# B&R Automation Studio project template1
Automation Studio 4.5.2.102

## Configuration Config1

### IoMap.iom - 4PP065_0571_P74/IoMap.iom
```iecst
VAR_CONFIG
	Cyclic#1.gAxis01_DrvIf.iLifeCnt AT %IB."8I64xxxxxxx.00x-1".SDC_LifeCnt;
	Cyclic#1.gAxis01_DrvIf.iDrvOK AT %IX."8I64xxxxxxx.00x-1".ETAD_Input_Bool_02;
	Cyclic#1.gAxis01_DrvIf.oSetTime AT %QW."8I64xxxxxxx.00x-1".SDC_SetTime;
	Cyclic#1.::speed AT %QW."8I64xxxxxxx.00x-1".LFRD_Output;
	Cyclic#1.gAxis01_DiDoIf.iLifeCntDriveReady AT %IB."8I64xxxxxxx.00x-1".SDC_LifeCnt;
	Cyclic#1.gAxis01_DiDoIf.iLifeCntDriveEnable AT %IB."8I64xxxxxxx.00x-1".SDC_LifeCnt;
	Cyclic#1.gAxis01_DiDoIf.oDriveEnable AT %QX."8I64xxxxxxx.00x-1".CMDD_Output_Bool_00;
	Cyclic#1.gAxis01_ModuleOk AT %QX."8I64xxxxxxx.00x-1".CMDD_Output_Bool_01;
	Cyclic#1.gAxis01_ModuleOk AT %QX."8I64xxxxxxx.00x-1".CMDD_Output_Bool_02;
	Cyclic#1.gAxis01_ModuleOk AT %IX."8I64xxxxxxx.00x-1".ModuleOk;
	Cyclic#1.gAxis01_DiDoIf.oDriveEnable AT %QX."8I64xxxxxxx.00x-1".CMDD_Output_Bool_03;
	Cyclic#1.gAxis01_DiDoIf.iDriveReady AT %IX."8I64xxxxxxx.00x-1".ETAD_Input_Bool_02;
	::EVIRD.STATE AT %IW."8I64xxxxxxx.00x-1".ETAD_Input;
	::EVIRD.CMD AT %QW."8I64xxxxxxx.00x-1".CMDD_Output;
	::led1 AT %QX."X20DO9322".DigitalOutput02;
	::led2 AT %QX."X20DO9322".DigitalOutput03;
	::led3 AT %QX."X20DO9322".DigitalOutput04;
	::led4 AT %QX."X20DO9322".DigitalOutput05;
	::real_speed AT %IW."8I64xxxxxxx.00x-1".RFRD_Input;
END_VAR
```

## Logical view

### Global.var
```iecst
VAR
	gAxis01 : ACP10AXIS_typ;
	gAxis01_HW : SdcHwCfg_typ := (0);
	gAxis01_DrvIf : SdcDrvIf16_typ := (0);
	gAxis01_DiDoIf : SdcDiDoIf_typ := (0);
	gAxis01_ModuleOk : BOOL := 0;
	speed : INT := 500;
	EVIRD : DRIVE;
	start : INT := 0;
	Button_1 : BOOL;
	led : ARRAY[0..3] OF BOOL;
	led4 : BOOL;
	led3 : BOOL;
	led2 : BOOL;
	led1 : BOOL;
	Button_3 : BOOL;
	Button_2 : BOOL;
	Button_4 : BOOL;
	real_speed : {REDUND_UNREPLICABLE} INT;
END_VAR
```

- Visualisation Logical/gAxis01obj/Visu (not shown)

### Library Logical/Libraries/Library

#### Library.fun
```iecst
{REDUND_ERROR} FUNCTION_BLOCK DRIVE (*TODO: Add your comment here*) (*$GROUP=User,$CAT=User,$GROUPICON=User.png,$CATICON=User.png*)
	VAR_INPUT
		ENABLED : BOOL;
		STATE : UINT;
	END_VAR
	VAR_OUTPUT
		CMD : UINT;
	END_VAR
END_FUNCTION_BLOCK
```

#### DRIVE.c
```c
#include <bur/plctypes.h>
#ifdef __cplusplus
	extern "C"
	{
#endif
	#include "Library.h"
#ifdef __cplusplus
	};
#endif
/* TODO: Add your comment here */
void DRIVE(struct DRIVE* inst)
{
	UINT mask= inst->STATE & 0x6f;
	if(!inst->ENABLED)
	{
		inst->CMD =CMD_SHUTDOWN;
	}
	else
	{
		switch(mask)
		{
			case STATE_DISABLED:
				inst->CMD=CMD_SHUTDOWN;
				break;
			case STATE_READY:
				inst->CMD=CMD_ENABLED;
				break;
			case STATE_SWITCHED_ON:
				inst->CMD=CMD_SWITCHED_ON;
				break;
		}
	}
}
```

### Program Logical/Program

#### Main.c
```c
#include <bur/plctypes.h>

#ifdef _DEFAULT_INCLUDES
#include <AsDefault.h>
#endif

void _INIT ProgramInit(void)
{
	real_speed=500;
	speed=500;
	EVIRD.ENABLED=1;
}

void _CYCLIC ProgramCyclic(void)
{
	DRIVE(&EVIRD);
	if(start == 1)  //Остановка двигателя если отжата кнопка Start
	{
		speed=0;
	}
	start =0;
	real_speed;
}

void _EXIT ProgramExit(void)
{

}
```

### Program Logical/Program1

#### Main.c
```c
#include <bur/plctypes.h>

#ifdef _DEFAULT_INCLUDES
	#include <AsDefault.h>
#endif

void _INIT ProgramInit(void)
{

}

void _CYCLIC ProgramCyclic(void)
{
	if(Button_1 ==1)
	{
		led[0]=!led[0];
		led[1]=led[1];
		led[2]=led[2];
		led[3]=!led[3];
		Button_1=!Button_1;
	}
	else if(Button_2 ==1)
	{
		Button_2=!Button_2;
		led[0]=!led[0];
		led[1]=!led[1];
		led[2]=led[2];
		led[3]=!led[3];
	}
	else if(Button_3 ==1)
	{
		Button_3=!Button_3;
		led[0]=!led[0];
		led[1]=!led[1];
		led[2]=!led[2];
		led[3]=led[3];
	}
	else if(Button_4 ==1)
	{
		Button_4=!Button_4;
		led[0]=led[0];
		led[1]=!led[1];
		led[2]=led[2];
		led[3]=!led[3];
	}
	led1=led[0];
	led2=led[1];
	led3=led[2];
	led4=led[3];

}

void _EXIT ProgramExit(void)
{

}
```

Listed in the project but not available here: Logical/gAxis01obj/gAxis01a, Logical/gAxis01obj/gAxis01i
